ABB RobotStudio station: Moja_prva_pick&place_stanica.rspag

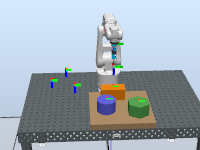
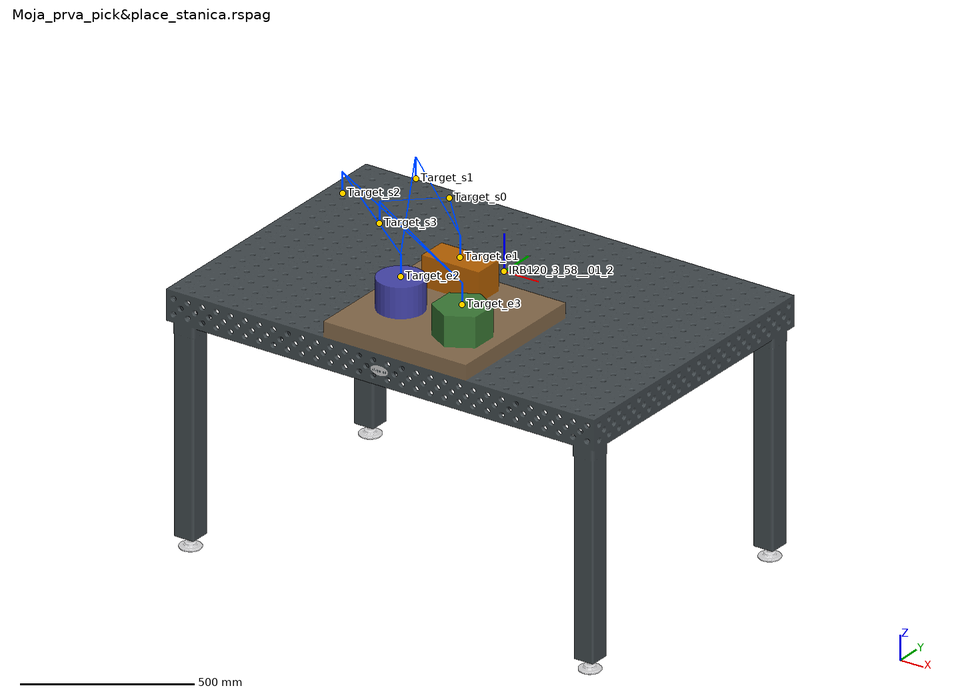
[picture v1: parts stored in the station drawn from their meshes, with robot base, taught points and paths (robot models come from the ABB library and are not in the file)]
--- station ---
Station Moja_prva_pick&place_stanica (saved by RobotStudio 21.4.9700.0)
Controller Controller1, task T_ROB1: task frame (RAPID world) sits at (0, 150, 830) mm, rotated rx 0 ry 0 rz -90 deg in the station
Controller Controller1
  mechanical unit ROB_1: IRB120_3_58__01_2, 6 joints, base frame (0, -20, 0) mm
Layout (positions relative to the parent item):
  - table [part] at (-200, -500, 830) mm, size 500 x 500 x 50 mm
  - object_1 [part] at (-200, -500, 830) mm, size 200 x 100 x 150 mm
  - object_2 [part] at (-200, -500, 830) mm, size 149.5 x 149.7 x 150 mm
  - object_3 [part] at (-200, -500, 830) mm, size 155.5 x 179.5 x 150 mm
  - siegmund_1500_1000 [part], size 1500 x 1010.3 x 830 mm
  - object_11 [part] at (-200, -500, 830) mm, size 200 x 100 x 150 mm
  - object_22 [part] at (-200, -500, 830) mm, size 149.5 x 149.7 x 150 mm
  - object_33 [part] at (-200, -500, 830) mm, size 155.5 x 179.5 x 150 mm
  - IRB120_3_58__01_2 [mechanism, from Robots\IRB120_3_58_G_01.rslib] at (-20, 150, 830) mm, rotated rx 0 ry 0 rz -90 deg; joint values [0.0661, 0.0025, -0.0025, 0, 1.5708, 0.0661] (rad or m)
  - smc_gripper [mechanism, from Veci_z_GitHubu\smc_gripper.rslib] at (0, -152, 1388) mm, rotated rx -180 ry 0 rz 90 deg
  - Positioner_3 [smart component, from Components\Positioner.rslib]
      properties: Object=object_1; Position=[-0.6 -0.15 0.83]; Orientation=[0 0 0]; Reference=Global; ReferenceObject=(none)
  - Attach_obj1 [smart component, from Components\Attacher.rslib]
      properties: Parent=smc_gripper; Flange=0; Child=object_1; Mount=false; Offset=[0 0 0]; Orientation=[0 0 0]
  - Detach_obj1 [smart component, from Components\Detacher.rslib]
      properties: Child=object_1; KeepPosition=true
  - Attach_obj2 [smart component, from Components\Attacher.rslib]
      properties: Parent=smc_gripper; Flange=0; Child=object_2; Mount=false; Offset=[0 0 0]; Orientation=[0 0 0]
  - Attach_obj3 [smart component, from Components\Attacher.rslib]
      properties: Parent=smc_gripper; Flange=0; Child=object_3; Mount=false; Offset=[0 0 0]; Orientation=[0 0 0]
  - Detach_obj3 [smart component, from Components\Detacher.rslib]
      properties: Child=object_3; KeepPosition=true
  - Positioner_4 [smart component, from Components\Positioner.rslib]
      properties: Object=object_2; Position=[-0.65 -0.15 0.83]; Orientation=[0 0 0]; Reference=Global; ReferenceObject=(none)
  - Positioner_5 [smart component, from Components\Positioner.rslib]
      properties: Object=object_3; Position=[-0.7 -0.2 0.83]; Orientation=[0 0 0]; Reference=Global; ReferenceObject=(none)
  - Detach_obj2 [smart component, from Components\Detacher.rslib]
      properties: Child=object_2; KeepPosition=true
  - LogicGate [smart component, from Components\LogicGate.rslib]
      properties: Operator=OR; Delay=0
  - LogicGate_2 [smart component, from Components\LogicGate.rslib]
      properties: Operator=OR; Delay=0
  - LogicGate_3 [smart component, from Components\LogicGate.rslib]
      properties: Operator=OR; Delay=0
Attachment: smc_gripper is attached to IRB120_3_58__01_2 / Link6
Station signals: DI Object_1_positioner
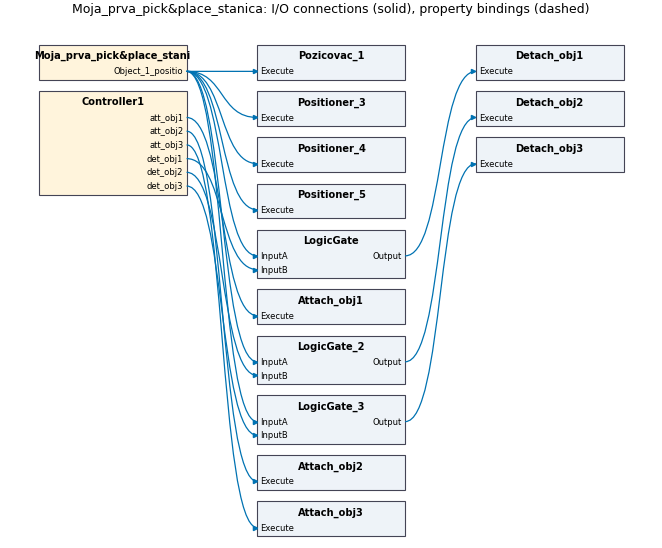
Station logic (signal -> signal, property => property):
  Moja_prva_pick&place_stanica.Object_1_positioner -> Pozicovac_1.Execute
  Moja_prva_pick&place_stanica.Object_1_positioner -> Positioner_3.Execute
  Controller1.att_obj1 -> Attach_obj1.Execute
  Controller1.att_obj2 -> Attach_obj2.Execute
  Controller1.att_obj3 -> Attach_obj3.Execute
  Moja_prva_pick&place_stanica.Object_1_positioner -> Positioner_4.Execute
  Moja_prva_pick&place_stanica.Object_1_positioner -> Positioner_5.Execute
  Moja_prva_pick&place_stanica.Object_1_positioner -> LogicGate_2.InputA
  Moja_prva_pick&place_stanica.Object_1_positioner -> LogicGate.InputA
  Moja_prva_pick&place_stanica.Object_1_positioner -> LogicGate_3.InputA
  LogicGate_3.Output -> Detach_obj3.Execute
  LogicGate_2.Output -> Detach_obj2.Execute
  LogicGate.Output -> Detach_obj1.Execute
  Controller1.det_obj1 -> LogicGate.InputB
  Controller1.det_obj2 -> LogicGate_2.InputB
  Controller1.det_obj3 -> LogicGate_3.InputB

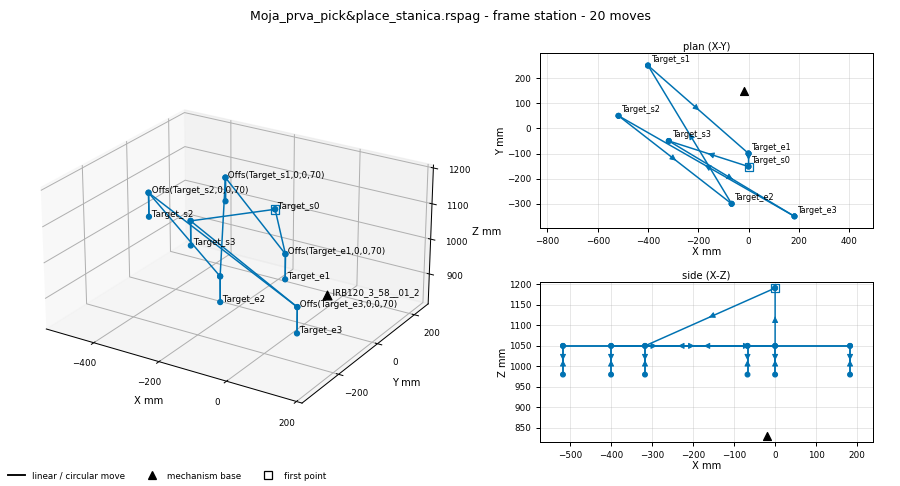
[picture p0: tool path of Moja_prva_pick&place_stanica.rspag in frame station, 20 of 20 moves have a stored position in this frame; points joined in program order, loops and branches not executed]
--- Backups/Controller1/RAPID/TASK1/PROGMOD/CalibData.mod ---
MODULE CalibData
    PERS tooldata smc_gripper:=[TRUE,[[0,0.004,197.001],[1,0,0,0]],[1,[0.207,-0.496,71.18],[1,0,0,0],0,0,0]];
ENDMODULE

--- Backups/Controller1/RAPID/TASK1/PROGMOD/Module1.mod ---
MODULE Module1
        CONST robtarget Target_s0:=[[302,0.004,360.999],[0,0,1,0],[-1,0,-1,0],[9E+09,9E+09,9E+09,9E+09,9E+09,9E+09]];
    CONST robtarget Target_s1:=[[-100,-400,150],[0,0,1,0],[-2,0,-2,0],[9E+09,9E+09,9E+09,9E+09,9E+09,9E+09]];
    CONST robtarget Target_e1:=[[250,0,150],[0,0,1,0],[-1,0,-1,0],[9E+09,9E+09,9E+09,9E+09,9E+09,9E+09]];
    CONST robtarget Target_s2:=[[100,-517.298,150],[0,0,1,0],[-1,0,-1,0],[9E+09,9E+09,9E+09,9E+09,9E+09,9E+09]];
    CONST robtarget Target_e2:=[[450,-67.298,150],[0,0,1,0],[-1,0,-1,0],[9E+09,9E+09,9E+09,9E+09,9E+09,9E+09]];
    CONST robtarget Target_s3:=[[200,-317.298,150],[0,0,1,0],[-1,0,-1,0],[9E+09,9E+09,9E+09,9E+09,9E+09,9E+09]];
    CONST robtarget Target_e3:=[[500,182.702,150],[0,0,1,0],[0,0,0,0],[9E+09,9E+09,9E+09,9E+09,9E+09,9E+09]];
    CONST robtarget Target_s0_2:=[[302,0.004,360.999],[0,0,1,0],[-1,0,-1,0],[9E+09,9E+09,9E+09,9E+09,9E+09,9E+09]];
!***********************************************************
    !
    ! Modul:  Module1
    !
    ! Popis:
    !   <Sem vlozte popis> A musim?
    !
    ! Autor: Pollak
    !
    ! Verze: 0.0.1
    !
    !***********************************************************


    !***********************************************************
    !
    ! Procedura main
    !
    !   Toto je vstupní bod vaseho programu
    !   Nene, toto je prva domaca uloha z VRM
    !***********************************************************
    PROC main()
        !Sem vlozte Vás kód
        !Dobre, tu je:
        Path_10;
        !passVRM()
    ENDPROC
    PROC Path_10()
        MoveL Target_s0,v100,fine,smc_gripper\WObj:=wobj0; !vychozia pozicia


        MoveL Offs(Target_s3, 0, 0, 70),v100,fine,smc_gripper\WObj:=wobj0; ! pohni sa ku targetu ale pridaj offset XYZ
        MoveL Target_s3,v100,fine,smc_gripper\WObj:=wobj0; ! pohni sa ku targetu
        PulseDO att_obj3; ! chyt objekt 3
        MoveL Offs(Target_s3, 0, 0, 70),v100,fine,smc_gripper\WObj:=wobj0; ! pohni sa ku targetu ale pridaj offset XYZ

        MoveL Offs(Target_e3, 0, 0, 70),v100,fine,smc_gripper\WObj:=wobj0; ! pohni sa ku targetu ale pridaj offset XYZ
        MoveL Target_e3,v100,fine,smc_gripper\WObj:=wobj0; ! pohni sa ku targetu
        PulseDO det_obj3; ! pust objekt 3
        WaitTime 1; ! cakaj
        MoveL Offs(Target_e3, 0, 0, 70),v100,fine,smc_gripper\WObj:=wobj0; ! pohni sa ku targetu ale pridaj offset XYZ


        MoveL Offs(Target_s2, 0, 0, 70),v100,fine,smc_gripper\WObj:=wobj0; ! pohni sa ku targetu ale pridaj offset XYZ
        MoveL Target_s2,v100,fine,smc_gripper\WObj:=wobj0; ! pohni sa ku targetu
        PulseDO att_obj2; ! chyt objekt 2
        MoveL Offs(Target_s2, 0, 0, 70),v100,fine,smc_gripper\WObj:=wobj0; ! pohni sa ku targetu ale pridaj offset XYZ

        MoveL Offs(Target_e2, 0, 0, 70),v100,fine,smc_gripper\WObj:=wobj0; ! pohni sa ku targetu ale pridaj offset XYZ
        MoveL Target_e2,v100,fine,smc_gripper\WObj:=wobj0; ! pohni sa ku targetu
        PulseDO det_obj2; ! pust objekt 2
        WaitTime 1; ! cakaj
        MoveL Offs(Target_e2, 0, 0, 70),v100,fine,smc_gripper\WObj:=wobj0; ! pohni sa ku targetu ale pridaj offset XYZ


        MoveL Offs(Target_s1, 0, 0, 70),v100,fine,smc_gripper\WObj:=wobj0; ! pohni sa ku targetu ale pridaj offset XYZ
        MoveL Target_s1,v100,fine,smc_gripper\WObj:=wobj0; ! pohni sa ku targetu
        PulseDO att_obj1; ! chyt objekt 1
        MoveL Offs(Target_s1, 0, 0, 70),v100,fine,smc_gripper\WObj:=wobj0; ! pohni sa ku targetu ale pridaj offset XYZ

        MoveL Offs(Target_e1, 0, 0, 70),v100,fine,smc_gripper\WObj:=wobj0; ! pohni sa ku targetu ale pridaj offset XYZ
        MoveL Target_e1,v100,fine,smc_gripper\WObj:=wobj0; ! pohni sa ku targetu
        PulseDO det_obj1; ! pust objekt 1
        WaitTime 1; ! cakaj
        MoveL Offs(Target_e1, 0, 0, 70),v100,fine,smc_gripper\WObj:=wobj0; ! pohni sa ku targetu ale pridaj offset XYZ


        MoveL Target_s0_2,v100,fine,smc_gripper\WObj:=wobj0; !vychozia pozicia
    ENDPROC
ENDMODULE

--- Backups/Controller1/SYSPAR/EIO.cfg ---
EIO:CFG_1.0:6:1::
#
EIO_SIGNAL:

      -Name "att_obj1" -SignalType "DO"

      -Name "det_obj1" -SignalType "DO"

      -Name "att_obj2" -SignalType "DO"

      -Name "att_obj3" -SignalType "DO"

      -Name "det_obj2" -SignalType "DO"

      -Name "det_obj3" -SignalType "DO"
